// TIA Portal V20 export
// export: Created 2025-12-01T14:56:13.9391558Z, ExportSetting None, DisplayName Totally Integrated Automation Portal, DisplayVersion V20 Update 3, DisplayName TIA Portal Openness, DisplayVersion V20 Update 3, DisplayName TIA Portal Version Control Interface, DisplayVersion V20 Update 3, DisplayName STEP 7 Professional, DisplayVersion V20 Update 3, DisplayName STEP 7 Safety, DisplayVersion V20 Update 2, DisplayName WinCC Basic/Comfort/Advanced, DisplayVersion V20 Update 3, DisplayName WinCC Professional, DisplayVersion V20 Update 3, DisplayName WinCC Unified, DisplayVersion V20 Update 3
TYPE "UDT_DatosDispositivo"
   STRUCT
      EstadoRecepcionEvento : UInt;   // Estado de la recepcion del Evento
      EstadoEmisionEvento : UInt;   // Estado de la Emision del Evento
      EstadoGeneralEvento : UInt;   // Estado general de los Eventos (Peticiones)
      EstadoOrdenDispo : UInt;   // Estado de la Orden enviada al Dispositivo
      EstadoPresenciaDispo : UInt;   // Estaod de la Presencia enviada del Dispositivo
      StatusActual : Word;   // Status actual del Dispositivo (Ultimo Evento)
      ErrorActual : UDInt;   // Error Actual del Dispositivo (Ultimo Evento)
      StatusReal : Word;   // Status Real del Dispositivo
      ErrorReal : UDInt;   // Error Real del Dispositivo
   END_STRUCT;
END_TYPE
